FUNCTION_BLOCK PACK_BYTE (* Packs 8 BOOLs into a BYTE *)
  (* Standard: 61499-1; Classification: Math *)
  (* Version 0.1, 2007-04-02, JHC, Holobloc Inc, Corrected type of OUT. *)
  (* Version 0.0, 2002-05-07, JHC, Rockwell Automation, Copied/Modified from PACK_WORD. *)
  (* Compiler header: package fb.rt.math; *)
  (* Compiler Java IBM VisualAge 3.0 *)
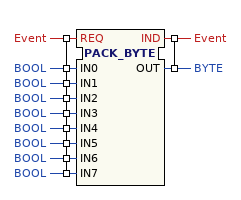
  EVENT_INPUT
    REQ WITH IN0, IN1, IN2, IN3, IN4, IN5, IN6, IN7; (* Pack Request *)
  END_EVENT
  EVENT_OUTPUT
    IND WITH OUT; (* Data Change Notification *)
  END_EVENT
  VAR_INPUT
    IN0 : BOOL; (* Data to Pack *)
    IN1 : BOOL;
    IN2 : BOOL;
    IN3 : BOOL;
    IN4 : BOOL;
    IN5 : BOOL;
    IN6 : BOOL;
    IN7 : BOOL;
  END_VAR
  VAR_OUTPUT
    OUT : BYTE; (* Packed Data *)
  END_VAR
  SERVICE APPLICATION/PACK_WORD
    SEQUENCE dataChanged
      APPLICATION.REQ(IN0,...,IN7) -> PACK_WORD.pack() -> APPLICATION.IND(OUT);
    END_SEQUENCE
    SEQUENCE dataUnchanged
      APPLICATION.REQ(IN0,...,IN7) -> PACK_WORD.pack();
    END_SEQUENCE
  END_SERVICE
END_FUNCTION_BLOCK
